// Mitsubishi GX Works2 project: MPS장비 TEST   PLC: Q03UDV

PROGRAM MAIN
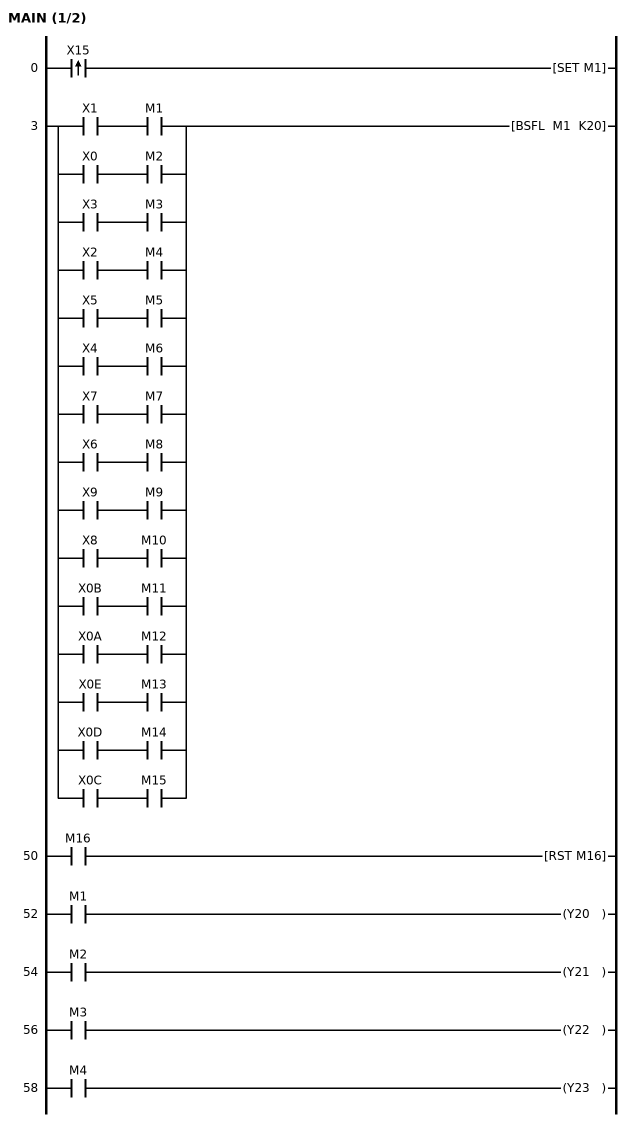
0     LDP     X15
      SET     M1
3     LD      X1
      AND     M1
      LD      X0
      AND     M2
      ORB
      LD      X3
      AND     M3
      ORB
      LD      X2
      AND     M4
      ORB
      LD      X5
      AND     M5
      ORB
      LD      X4
      AND     M6
      ORB
      LD      X7
      AND     M7
      ORB
      LD      X6
      AND     M8
      ORB
      LD      X9
      AND     M9
      ORB
      LD      X8
      AND     M10
      ORB
      LD      X0B
      AND     M11
      ORB
      LD      X0A
      AND     M12
      ORB
      LD      X0E
      AND     M13
      ORB
      LD      X0D
      AND     M14
      ORB
      LD      X0C
      AND     M15
      ORB
      BSFL    M1 K20
50    LD      M16
      RST     M16
52    LD      M1
      OUT     Y20
54    LD      M2
      OUT     Y21
56    LD      M3
      OUT     Y22
58    LD      M4
      OUT     Y23
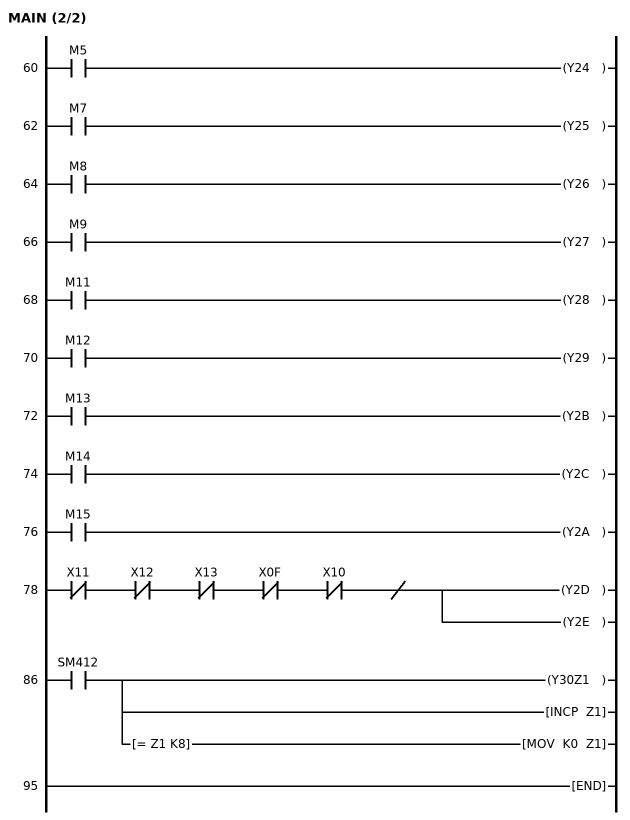
60    LD      M5
      OUT     Y24
62    LD      M7
      OUT     Y25
64    LD      M8
      OUT     Y26
66    LD      M9
      OUT     Y27
68    LD      M11
      OUT     Y28
70    LD      M12
      OUT     Y29
72    LD      M13
      OUT     Y2B
74    LD      M14
      OUT     Y2C
76    LD      M15
      OUT     Y2A
78    LDI     X11
      ANI     X12
      ANI     X13
      ANI     X0F
      ANI     X10
      INV
      OUT     Y2D
      OUT     Y2E
86    LD      SM412
      OUT     Y30Z1
      INCP    Z1
      AND=    Z1 K8
      MOV     K0 Z1
95    END
END_PROGRAM
